(* Logix 5000 project; controller CancelaAutomotivaParte1 vendor 1 type 14 code 89 rev 20.12; software revision 20.04 *)

TASK MainTask (continuous, watchdog 500 ms) : MainProgram

MODULES
   Controller : vendor 1 type 14 code 89 (CompactLogixL23E_QBFC1_Controller 0, rev 20.12)
      LocalENB : vendor 1 type 12 code 191 (CompactLogixL23E_QBFC1_Ethernet 1, rev 20.11)
      Local : CompactBus (CompactVirtualAdapter 3, rev 20.11)
         Discrete_Inputs : vendor 1 type 7 code 320 (Compact 1, rev 3.1, Input RPI 20 ms)
         Discrete_Outputs : vendor 1 type 7 code 322 (Compact 2, rev 3.1, Output RPI 20 ms)
         Analog_IO : vendor 1 type 10 code 120 (Compact 3, rev 1.1, Output RPI 80 ms)
         Counters : vendor 1 type 109 code 70 (Compact 4, rev 1.1, Output RPI 20 ms)
END_MODULES

PROGRAM MainProgram   (* main routine MainRoutine *)
VAR
   AbrirCancela : ALIAS FOR Local:2:O.Data.1;
   AcessoPermitido : BOOL;
   ArrecadTotal : DINT;
   BDPresCar : BOOL;
   CarPag : COUNTER;
   CarPas : COUNTER;
   CarroPassando : BOOL;
   ChamaContCarPag : BOOL;
   ChamaContCarPas : BOOL;
   Despesas : DINT;
   DespesaTotal : DINT;
   Entradas : DINT;
   espera500 : TIMER := (PRE := 500);
   FecharCancela : ALIAS FOR Local:2:O.Data.2;
   LeituraCracha : ALIAS FOR Local:1:I.Data.1;
   Lucro : DINT;
   LucroNegativo : BOOL;
   LucroPositivo : BOOL;
   Minuto : TIMER := (PRE := 60000);
   PresencaCarro : ALIAS FOR Local:1:I.Data.4;
   SePagando : BOOL;
   StartStop : ALIAS FOR Local:1:I.Data.3;
   TempoDescida : TIMER := (PRE := 5000);
   TempoEspera : TIMER := (PRE := 10000);
   TempoSubida : TIMER := (PRE := 5000);
   TotalizadorMinutos : COUNTER;
END_VAR

ROUTINE Arrecadacao   (* ladder *)
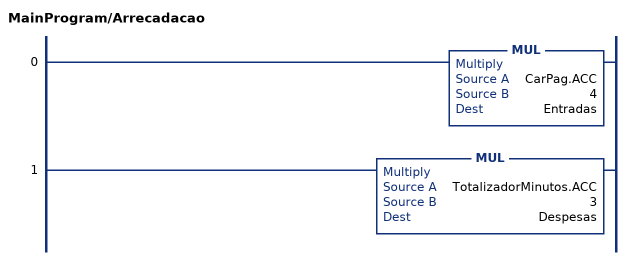
   0: MUL(CarPag.ACC,4,Entradas);
   1: MUL(TotalizadorMinutos.ACC,3,Despesas);
END_ROUTINE

ROUTINE ContCarPag   (* ladder *)
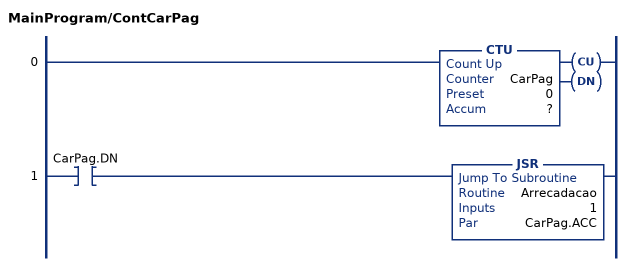
   0: CTU(CarPag,?,?);
   1: XIC(CarPag.DN)JSR(Arrecadacao,1,CarPag.ACC);
END_ROUTINE

ROUTINE ContCarPas   (* ladder *)
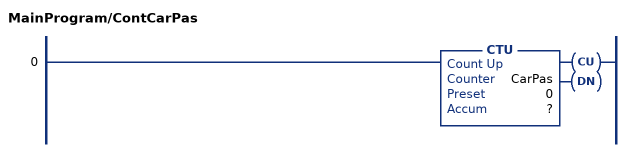
   0: CTU(CarPas,?,?);
END_ROUTINE

ROUTINE MainRoutine   (* ladder *)
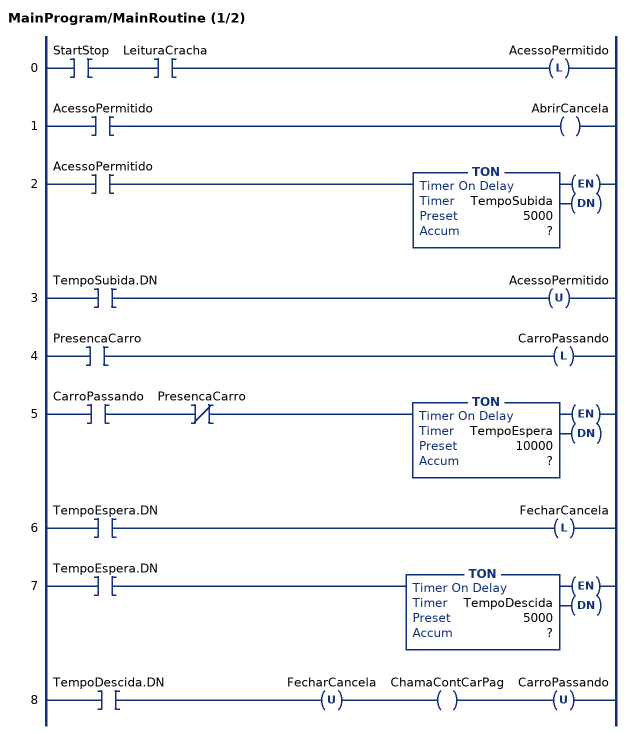
   0: XIC(StartStop)XIC(LeituraCracha)OTL(AcessoPermitido);
   1: XIC(AcessoPermitido)OTE(AbrirCancela);
   2: XIC(AcessoPermitido)TON(TempoSubida,?,?);
   3: XIC(TempoSubida.DN)OTU(AcessoPermitido);
   4: XIC(PresencaCarro)OTL(CarroPassando);
   5: XIC(CarroPassando)XIO(PresencaCarro)TON(TempoEspera,?,?);
   6: XIC(TempoEspera.DN)OTL(FecharCancela);
   7: XIC(TempoEspera.DN)TON(TempoDescida,?,?);
   8: XIC(TempoDescida.DN)OTU(FecharCancela)OTE(ChamaContCarPag)OTU(CarroPassando);
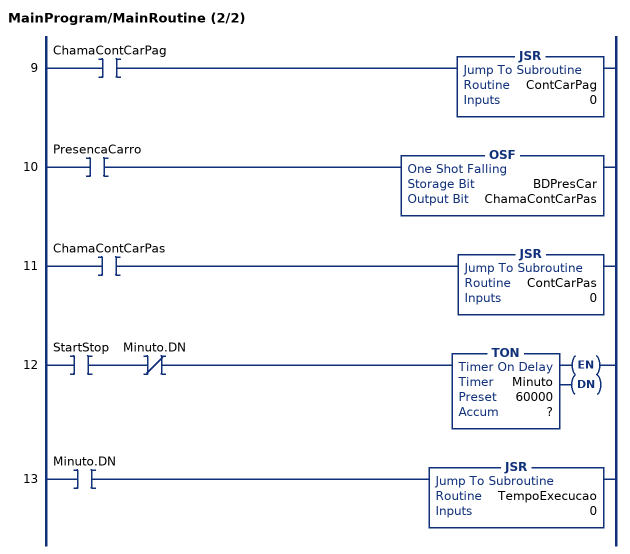
   9: XIC(ChamaContCarPag)JSR(ContCarPag,0);
   10: XIC(PresencaCarro)OSF(BDPresCar,ChamaContCarPas);
   11: XIC(ChamaContCarPas)JSR(ContCarPas,0);
   12: XIC(StartStop)XIO(Minuto.DN)TON(Minuto,?,?);
   13: XIC(Minuto.DN)JSR(TempoExecucao,0);
END_ROUTINE

ROUTINE Rentabilidade   (* ladder *)
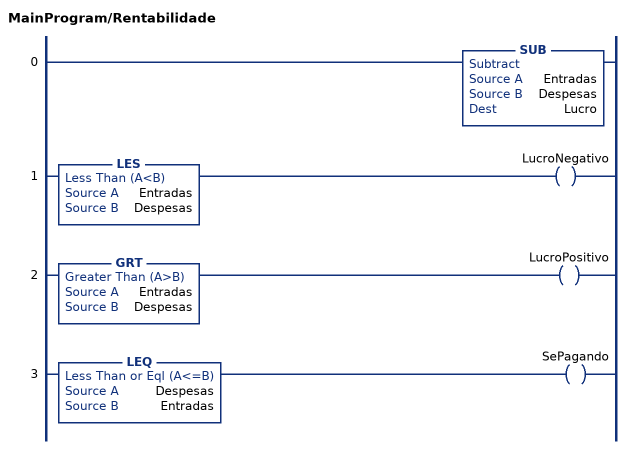
   0: SUB(Entradas,Despesas,Lucro);
   1: LES(Entradas,Despesas)OTE(LucroNegativo);
   2: GRT(Entradas,Despesas)OTE(LucroPositivo);
   3: LEQ(Despesas,Entradas)OTE(SePagando);
END_ROUTINE

ROUTINE TempoExecucao   (* ladder *)
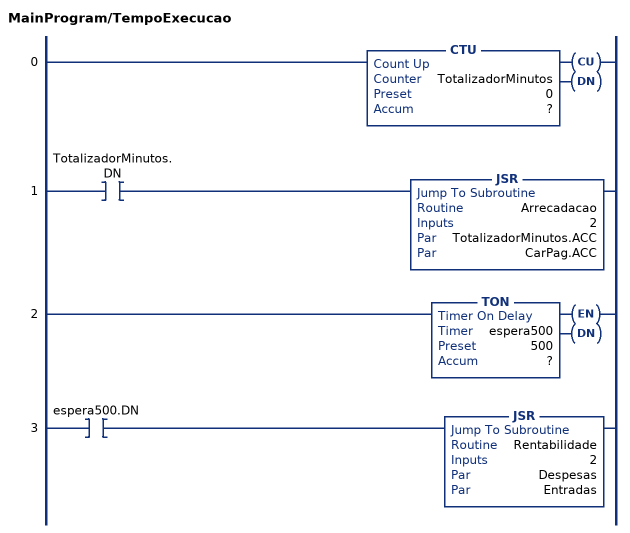
   0: CTU(TotalizadorMinutos,?,?);
   1: XIC(TotalizadorMinutos.DN)JSR(Arrecadacao,2,TotalizadorMinutos.ACC,CarPag.ACC);
   2: TON(espera500,?,?);
   3: XIC(espera500.DN)JSR(Rentabilidade,2,Despesas,Entradas);
END_ROUTINE
END_PROGRAM
